FUNCTION_BLOCK PowerOn
VAR_INPUT
	iControl_on  	: BOOL;
	iControl_off    : BOOL;
	iAuto_Man 		: BOOL;
	iEMRSTOP		: bool;
END_VAR
VAR_OUTPUT
	 ENO    : BOOL;
	qPower_On	 : BOOL;
	qStnAuto	 :BOOL;
	qStnMan  	 : BOOL;
END_VAR
VAR	
END_VAR

// Control ON Logic
IF iControl_On AND NOT iControl_off AND (Stn710_DB.Alarm_count = 0 OR Stn710_DB.Alarm_count > 1)  THEN
	qPower_On := TRUE;	
	ELSE
	qPower_On := FALSE;
END_IF

// Auto Logic
IF qPower_On AND NOT iAuto_Man THEN
	qStnAuto := TRUE;
	qStnMan := FALSE;
	ELSE
	qStnAuto := FALSE;	
END_IF
// Manual Logic
IF qPower_On AND iAuto_Man THEN
	qStnMan := TRUE;
	qStnAuto := FALSE;
	
	ELSE
	qStnMan := FALSE;	
END_IF

END_FUNCTION_BLOCK

(* stored: Version 1.1.0.1, ProductVersion 3.1.4024.16
   POU PowerOn: Id {b732c427-247d-4a1e-854c-17af1c115c65}, SpecialFunc None *)
